TYPE ST_InterMachineCom_SlaveConData :
STRUCT
	enable			: BOOL;
	BrokerIP		: STRING;
END_STRUCT
END_TYPE

(* stored: Version 1.1.0.1, ProductVersion 3.1.4026.18
   DUT ST_InterMachineCom_SlaveConData: Id {bd1409f7-dec6-4c13-8935-fe58e5b0011f} *)
